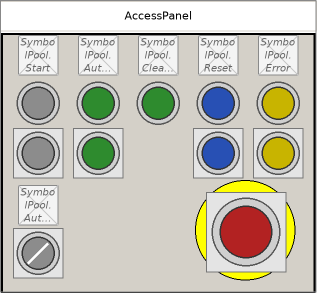
VISUALIZATION V_AccessPanel  // 317x293
VAR_IN_OUT
	Signals  : ST_AccessPanel;
END_VAR
    Rectangle (1,33 314x260)
    Image (18,35 40x40), image: SymbolPool.Start
    PushSwitch (13,128 50x50), tooltip "Activate main contactor", variable: Signals.inputs.PB_ActivateMainContactor, behaviour: TAP, style: Switch-PushSwitch-Gray
    Lamp1 (13,78 50x50), tooltip "Main contactor activated", variable: Signals.outputs.LED_MainContactorActivated, style: Lamp-Lamp1-Gray
    PushSwitch (73,128 50x50), tooltip "Auto on", variable: Signals.inputs.PB_AutoOn, behaviour: TAP, style: Switch-PushSwitch-Green
    Lamp1 (73,78 50x50), tooltip "Auto activated", variable: Signals.outputs.LED_AutoIsOn, style: Lamp-Lamp1-Green
    Lamp1 (133,78 50x50), tooltip "Clear enterance", variable: Signals.outputs.LED_ClearEnterance, style: Lamp-Lamp1-Green
    Lamp1 (193,78 50x50), tooltip "Emergency stop", variable: Signals.outputs.LED_EmergencyStop, style: Lamp-Lamp1-Blue
    PushSwitch (193,128 50x50), tooltip "Reset emergency stop", variable: Signals.inputs.PB_EmergencyStopReset, behaviour: TAP, style: Switch-PushSwitch-Blue
    Lamp1 (253,78 50x50), tooltip "Error", variable: Signals.outputs.LED_Error, style: Lamp-Lamp1-Yellow
    PushSwitch (253,128 50x50), tooltip "Reset error", variable: Signals.inputs.PB_ErrorReset, behaviour: TAP, style: Switch-PushSwitch-Yellow
    RotarySwitch (13,228 50x50), tooltip "Auto/Entry request key switch", variable: Signals.inputs.SW_EntryRequest, behaviour: TOGGLE, style: Switch-RotarySwitch-Gray
    Ellipse (195,180 100x100)
    PushSwitch (206,192 80x80), variable: Signals.inputs.PB_EmergencyStop, behaviour: TOGGLE, style: Switch-PushSwitch-Red
    Image (78,35 40x40), image: SymbolPool.AutoOn
    Image (138,35 40x40), image: SymbolPool.ClearToEnter
    Image (198,35 40x40), image: SymbolPool.Reset
    Image (258,35 40x40), image: SymbolPool.Error
    Image (18,185 40x40), image: SymbolPool.AutoMan
    Textfield (0,1 317x30), "AccessPanel"
END_VISUALIZATION

(* stored: Version 1.1.0.1, ProductVersion 3.1.4024.4
   Visu V_AccessPanel: Id {b8513725-af41-40da-99a7-a6b5d411c619} *)
